// TIA Portal V21 export
FUNCTION "__PI_CREATEFC_NAME__" : Void   // FC__PI_CREATEFC_NUMBER__, SCL
{ S7_Optimized_Access := 'TRUE' }
// Minimal disposable SCL FC template imported by TiaLocalBridge.
// stored: IsIECCheckEnabled true, SetENOAutomatically true
BEGIN
   REGION Generated template
     //Minimal FC template created by TiaLocalBridge.
   END_REGION Generated template
END_FUNCTION
